PROGRAM MAIN
VAR
END_VAR

END_PROGRAM

(* stored: Version 1.1.0.1
   POU MAIN: Id {3e8ee53b-4ba3-40a1-bc6e-e2aed8eb2a14} *)
